// Verifies if a pressure (TORR) is near atmospheric pressure
FUNCTION F_Atm : BOOL
VAR_INPUT
	fPressure : REAL;
END_VAR
VAR
END_VAR

// Check that fPressure is within our error range for atmospheric pressure
F_Atm := ABS(ATM_PRESS - fPressure) <= ATM_PRESS_ERR_RNG;

END_FUNCTION

(* stored: Version 1.1.0.1, ProductVersion 3.1.4024.0
   POU F_Atm: Id {79f6dbdc-f5aa-4b39-b5b3-c2f56ea5db42}, SpecialFunc None *)
